TYPE st_BMS_Get :
STRUCT
	BatteryInfo							: st_BMS_BatterySummary;
	
	T_RemainingTimeToAutoCalibration	: TIME;
	

	//detailed info	
	MBMU								:	st_MBMU_Status;
	SBMU								:	ARRAY[0..3] OF st_SBMU_Status;
	
	Events								:	st_BMS_Events;
END_STRUCT
END_TYPE

(* stored: Version 1.1.0.1, ProductVersion 3.1.4024.12
   DUT st_BMS_Get: Id {005a8443-595a-4537-b6a8-503255910a5e} *)
